// TIA Portal V20 export
TYPE "LER_typeHotWireCutterInterface"
// stored: Access Published
   STRUCT
      commands : "LER_typeHotWireCutterCommands";
      monitoring : "LER_typeHotWireCutterMonitoring";
   END_STRUCT;
END_TYPE
